// TIA Portal V18 export
FUNCTION_BLOCK "_ML2_ts_block1"   // FB49, FBD
{ S7_Optimized_Access := 'TRUE' }
VERSION : 0.1
// stored: AutoNumber true, IsIECCheckEnabled false, IsRetainMemResEnabled false, MemoryReserve 100, SetENOAutomatically false, UDAEnableTagReadback false
   VAR_INPUT
      R_ALL : Bool;
      SwAuto : Bool;
      AutoRuning : Bool;
      Arrived : Bool;
      R_SeimAuto : Bool;
      CLK_Spot : Bool;
      CLK_Defect : Bool;
      CLK_Home : Bool;
      CLK_Load : Bool;
      CLK_Control2 : Bool;
      CLK_Control1 : Bool;
   END_VAR
   VAR_OUTPUT
      Q0_Auto : Bool;
      q0_AutoWaiting : Bool;
      Q0_SemiAuto : Bool;
      P1_Spot : Bool;
      Q1_Spot : Bool;
      P2_Defect : Bool;
      Q2_Defect : Bool;
      P3_Home : Bool;
      Q3_Home : Bool;
      P4_Load : Bool;
      Q4_Load : Bool;
      P5_Control1 : Bool;
      Q5_Control1 : Bool;
      P6_Control2 : Bool;
      Q6_control2 : Bool;
      Q99_none : Bool;
      Q99_Any : Bool;
   END_VAR
   VAR
      memarrived : Bool;
      reset_Qs : Bool;
      last_button_stands_Instance { S7_SetPoint := 'True'} : "last_button_stands";
      Q_integer { S7_SetPoint := 'True'} : Int;
      trDefect { S7_SetPoint := 'True'} : R_TRIG;
      trSpot { S7_SetPoint := 'True'} : R_TRIG;
      bsu_Spot { S7_SetPoint := 'True'} : "_ML2_ts_block1_subunit";
      bsu_Defect { S7_SetPoint := 'True'} : "_ML2_ts_block1_subunit";
      bsuHome { S7_SetPoint := 'True'} : "_ML2_ts_block1_subunit";
      bsu_load { S7_SetPoint := 'True'} : "_ML2_ts_block1_subunit";
      bsuControl1 { S7_SetPoint := 'True'} : "_ML2_ts_block1_subunit";
      bsuControl2 { S7_SetPoint := 'True'} : "_ML2_ts_block1_subunit";
   END_VAR
   VAR CONSTANT
      Qi0_off : Int := 0;
      Qi1_Spot : Int := 1;
      Qi2_Defect : Int := 2;
      Qi3Home : Int := 3;
      Qi4Load : Int := 4;
      Qi5Control1 : Int := 5;
      Qi6Control2 : Int := 6;
   END_VAR
   VAR_TEMP   // added for the SCL form of the ladder/FBD networks
      _w1 : Bool;
   END_VAR
BEGIN

REGION Network 2
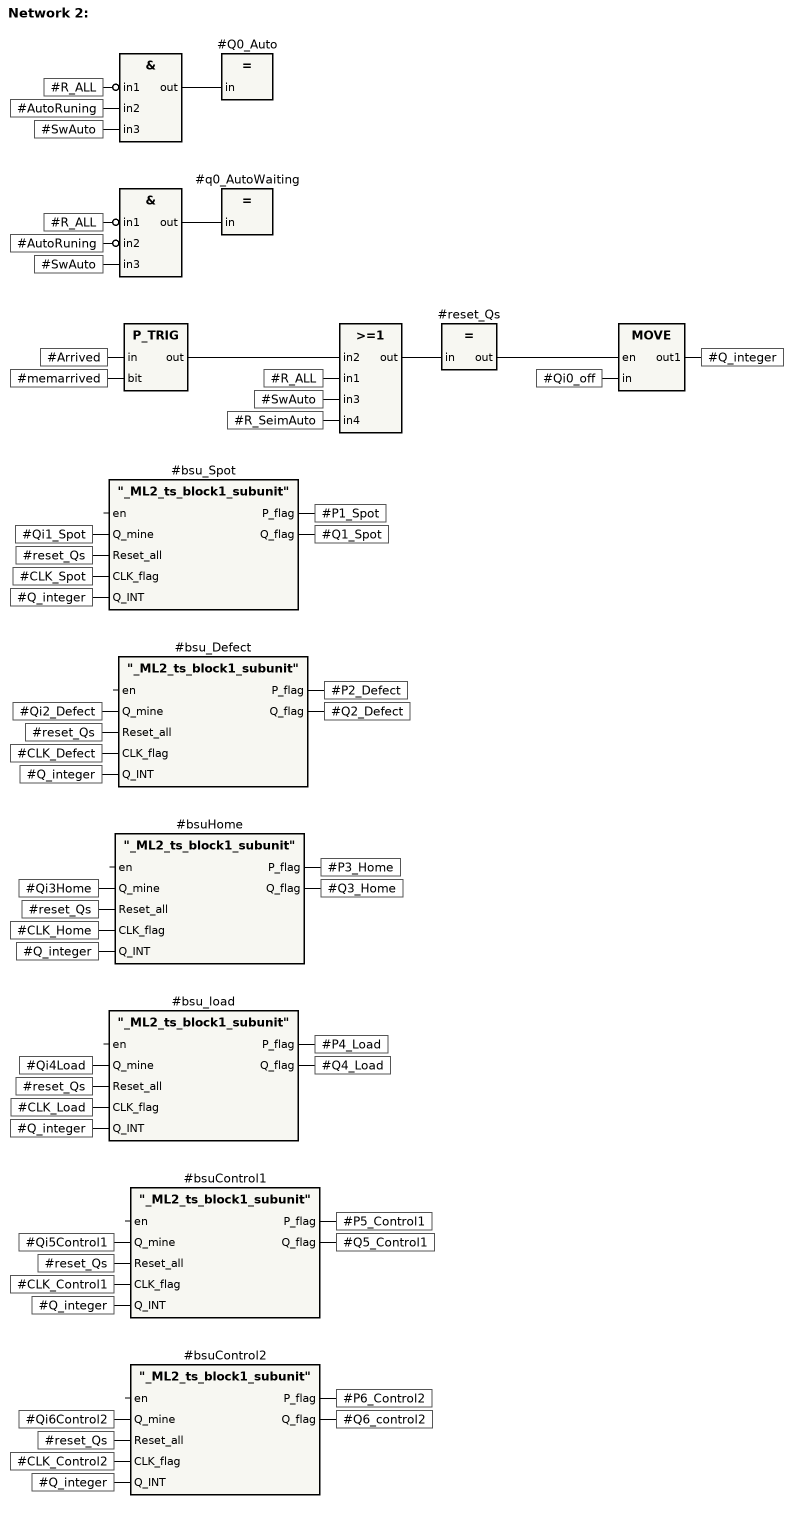
   #Q0_Auto := NOT #R_ALL AND #AutoRuning AND #SwAuto;
   #q0_AutoWaiting := NOT #R_ALL AND NOT #AutoRuning AND #SwAuto;
   #_w1 := #Arrived AND NOT #memarrived;   // rising edge
   #memarrived := #Arrived;
   #reset_Qs := #_w1 OR #R_ALL OR #SwAuto OR #R_SeimAuto;
   IF #reset_Qs THEN #Q_integer := #Qi0_off; END_IF;
   #bsu_Spot(Q_mine := #Qi1_Spot,   // "_ML2_ts_block1_subunit"
             Reset_all := #reset_Qs,
             CLK_flag := #CLK_Spot,
             Q_INT := #Q_integer,
             P_flag => #P1_Spot,
             Q_flag => #Q1_Spot);
   #bsu_Defect(Q_mine := #Qi2_Defect,   // "_ML2_ts_block1_subunit"
               Reset_all := #reset_Qs,
               CLK_flag := #CLK_Defect,
               Q_INT := #Q_integer,
               P_flag => #P2_Defect,
               Q_flag => #Q2_Defect);
   #bsuHome(Q_mine := #Qi3Home,   // "_ML2_ts_block1_subunit"
            Reset_all := #reset_Qs,
            CLK_flag := #CLK_Home,
            Q_INT := #Q_integer,
            P_flag => #P3_Home,
            Q_flag => #Q3_Home);
   #bsu_load(Q_mine := #Qi4Load,   // "_ML2_ts_block1_subunit"
             Reset_all := #reset_Qs,
             CLK_flag := #CLK_Load,
             Q_INT := #Q_integer,
             P_flag => #P4_Load,
             Q_flag => #Q4_Load);
   #bsuControl1(Q_mine := #Qi5Control1,   // "_ML2_ts_block1_subunit"
                Reset_all := #reset_Qs,
                CLK_flag := #CLK_Control1,
                Q_INT := #Q_integer,
                P_flag => #P5_Control1,
                Q_flag => #Q5_Control1);
   #bsuControl2(Q_mine := #Qi6Control2,   // "_ML2_ts_block1_subunit"
                Reset_all := #reset_Qs,
                CLK_flag := #CLK_Control2,
                Q_INT := #Q_integer,
                P_flag => #P6_Control2,
                Q_flag => #Q6_control2);
END_REGION

REGION Network 3
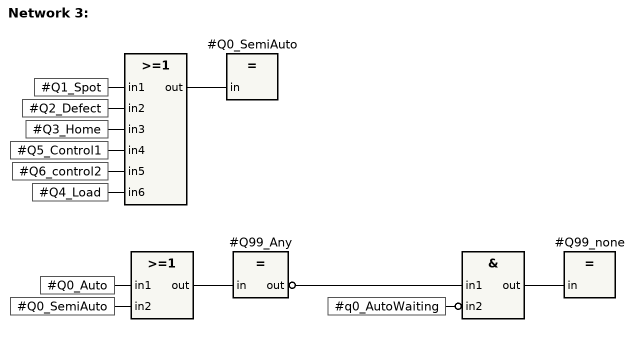
   #Q0_SemiAuto := #Q1_Spot OR #Q2_Defect OR #Q3_Home OR #Q5_Control1 OR #Q6_control2 OR #Q4_Load;
   #_w1 := #Q0_Auto OR #Q0_SemiAuto;
   #Q99_Any := #_w1;
   #Q99_none := NOT #_w1 AND NOT #q0_AutoWaiting;
END_REGION
END_FUNCTION_BLOCK
